// Mitsubishi GX Works2 project: inverter-1   PLC: Q03UDV

PROGRAM SPINDRY
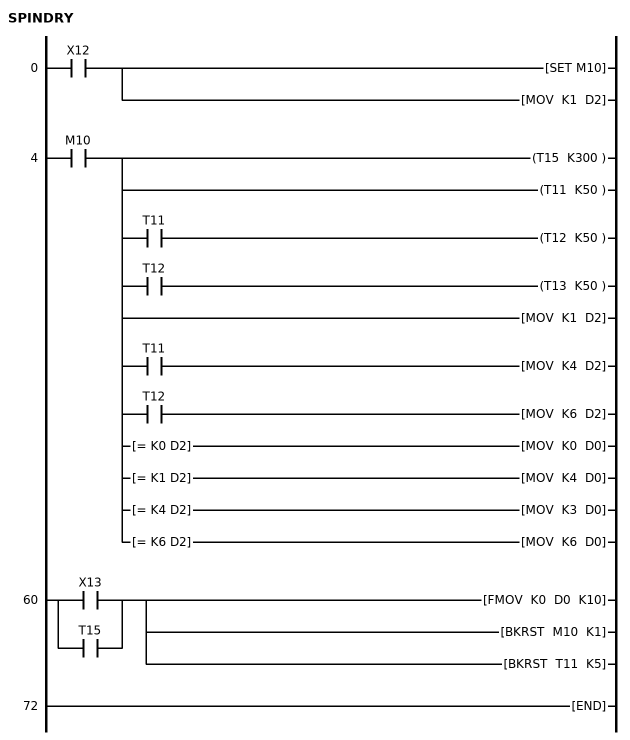
0     LD      X12
      SET     M10
      MOV     K1 D2
4     LD      M10
      OUT     T15 K300
      OUT     T11 K50
      MPS
      AND     T11
      OUT     T12 K50
      MRD
      AND     T12
      OUT     T13 K50
      MPP
      MOV     K1 D2
      MPS
      AND     T11
      MOV     K4 D2
      MRD
      AND     T12
      MOV     K6 D2
      MRD
      AND=    K0 D2
      MOV     K0 D0
      MRD
      AND=    K1 D2
      MOV     K4 D0
      MRD
      AND=    K4 D2
      MOV     K3 D0
      MPP
      AND=    K6 D2
      MOV     K6 D0
60    LD      X13
      OR      T15
      FMOV    K0 D0 K10
      BKRST   M10 K1
      BKRST   T11 K5
72    END
END_PROGRAM

PROGRAM BASIC
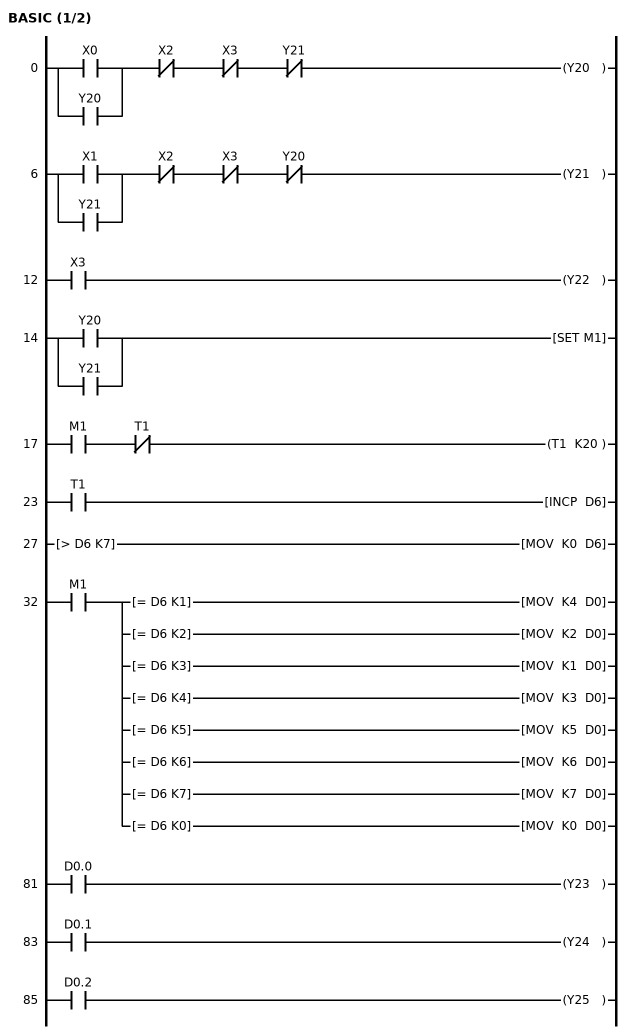
0     LD      X0
      OR      Y20
      ANI     X2
      ANI     X3
      ANI     Y21
      OUT     Y20
6     LD      X1
      OR      Y21
      ANI     X2
      ANI     X3
      ANI     Y20
      OUT     Y21
12    LD      X3
      OUT     Y22
14    LD      Y20
      OR      Y21
      SET     M1
17    LD      M1
      ANI     T1
      OUT     T1 K20
23    LD      T1
      INCP    D6
27    LD>     D6 K7
      MOV     K0 D6
32    LD      M1
      MPS
      AND=    D6 K1
      MOV     K4 D0
      MRD
      AND=    D6 K2
      MOV     K2 D0
      MRD
      AND=    D6 K3
      MOV     K1 D0
      MRD
      AND=    D6 K4
      MOV     K3 D0
      MRD
      AND=    D6 K5
      MOV     K5 D0
      MRD
      AND=    D6 K6
      MOV     K6 D0
      MRD
      AND=    D6 K7
      MOV     K7 D0
      MPP
      AND=    D6 K0
      MOV     K0 D0
81    LD      D0.0
      OUT     Y23
83    LD      D0.1
      OUT     Y24
85    LD      D0.2
      OUT     Y25
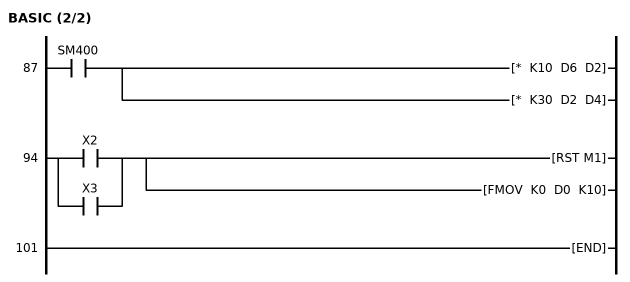
87    LD      SM400
      *       K10 D6 D2
      *       K30 D2 D4
94    LD      X2
      OR      X3
      RST     M1
      FMOV    K0 D0 K10
101   END
END_PROGRAM

PROGRAM HMI
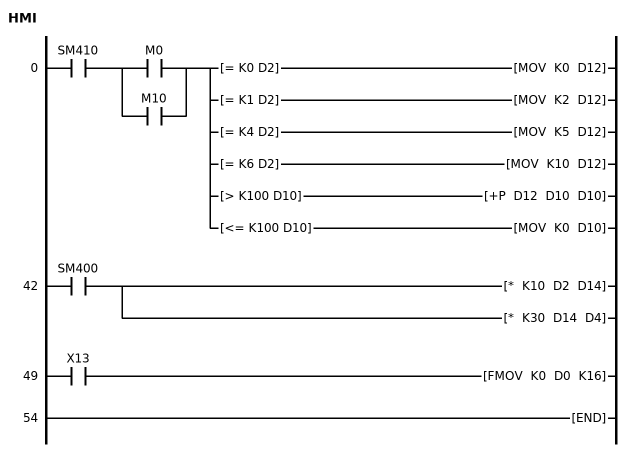
0     LD      SM410
      LD      M0
      OR      M10
      ANB
      MPS
      AND=    K0 D2
      MOV     K0 D12
      MRD
      AND=    K1 D2
      MOV     K2 D12
      MRD
      AND=    K4 D2
      MOV     K5 D12
      MRD
      AND=    K6 D2
      MOV     K10 D12
      MRD
      AND>    K100 D10
      +P      D12 D10 D10
      MPP
      AND<=   K100 D10
      MOV     K0 D10
42    LD      SM400
      *       K10 D2 D14
      *       K30 D14 D4
49    LD      X13
      FMOV    K0 D0 K16
54    END
END_PROGRAM

PROGRAM WASHER
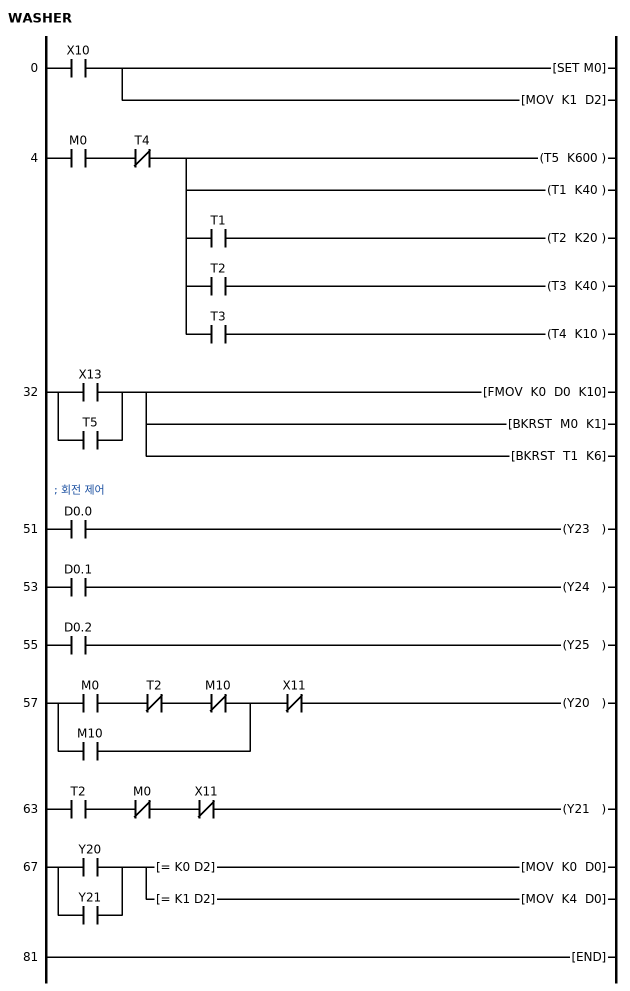
0     LD      X10
      SET     M0
      MOV     K1 D2
4     LD      M0
      ANI     T4
      OUT     T5 K600
      OUT     T1 K40
      MPS
      AND     T1
      OUT     T2 K20
      MRD
      AND     T2
      OUT     T3 K40
      MPP
      AND     T3
      OUT     T4 K10
32    LD      X13
      OR      T5
      FMOV    K0 D0 K10
      BKRST   M0 K1
      BKRST   T1 K6
; 회전 제어
51    LD      D0.0
      OUT     Y23
53    LD      D0.1
      OUT     Y24
55    LD      D0.2
      OUT     Y25
57    LD      M0
      ANI     T2
      ANI     M10
      OR      M10
      ANI     X11
      OUT     Y20
63    LD      T2
      ANI     M0
      ANI     X11
      OUT     Y21
67    LD      Y20
      OR      Y21
      MPS
      AND=    K0 D2
      MOV     K0 D0
      MPP
      AND=    K1 D2
      MOV     K4 D0
81    END
END_PROGRAM
